PROGRAM MAIN
VAR
	zmienna : INT;
	
END_VAR

END_PROGRAM

(* stored: Version 1.1.0.1, ProductVersion 3.1.4024.2
   POU MAIN: Id {b8de5909-2768-46d4-b7e1-95ca8e910a66}, SpecialFunc None *)
